FUNCTION_BLOCK TcoQl355P_v_1_x_x EXTENDS TcoCore.TcoComponent
VAR_INPUT
END_VAR
VAR_OUTPUT
END_VAR
VAR
    {attribute addProperty Name "<#Status#>"}
    _status : TcoQlSeriesSupply_Status_v_1_x_x;
    {attribute addProperty Name "<#Config#>"}
    _config : TcoQlSeriesSupply_Config_v_1_x_x;
    _someTaskIsActive : BOOL;
END_VAR
VAR
    {attribute addProperty Name "<#Get Command#>"}
    _getCommandTask : TcoQlGetCommandTask(THIS^);
    {attribute addProperty Name "<#Set Command#>"}
    _setCommandTask : TcoQlSetCommandTask(THIS^);
    {attribute addProperty Name "<#Restore#>"}
    _restoreTask : TcoCore.TcoTask(THIS^);
END_VAR
VAR
    {attribute 'hide'}
    _sb : TcoCore.StringBuilder;
END_VAR

_getCommandTask(inoConfig := _config, inoStatus := _status);
_setCommandTask(inoConfig := _config, inoStatus := _status);
//*************RESTORE********************
_restoreTask.Enabled := TRUE;

IF _restoreTask.Execute() THEN
    Restore();
    _restoreTask.DoneWhen(TRUE);
    _status.ActionDescription := 'Restored';
END_IF
//****************************************

(*~
    <docu>
        <summary>
            Gets the configuration of the IRC 5.
        </summary>
    </docu>
~*)
PROPERTY Config : REFERENCE TO TcoQlSeriesSupply_Config_v_1_x_x
GET
Config REF= _config;
END_GET
END_PROPERTY

METHOD FB_init : BOOL
VAR_INPUT
    bInitRetains : BOOL; // if TRUE, the retain variables are initialized (warm start / cold start)
    bInCopyCode : BOOL; // if TRUE, the instance afterwards gets moved into the copy code (online change)
    ParentObject : ITcoObject;
END_VAR
END_METHOD

METHOD PUBLIC GetCommand : TcoCore.ITcoTaskStatus
VAR_INPUT
    inCommand : TcoQlSeriesSupply_getControl_v_1_x_x;
END_VAR
GetCommand := _getCommandTask.WithParams(inCommand).Invoke();
END_METHOD

PROPERTY GetCommandTask : TcoCore.ITcoTaskStatus
GET
GetCommandTask := _getCommandTask;
END_GET
END_PROPERTY

METHOD PUBLIC GetCurrent : TcoCore.ITcoTaskStatus
VAR_INPUT
    (*~
    <docu>
        <summary>
            The number of the output or status register to which the command relates.
            Note that on single output supplies <N>=1 always.
            Note also that <N>= 3 refers to the AUX output. The AUX output has limited remote control functionality.
            For clarity, the commands where <N>= 3 can be used are explicitly commented; elsewhere only <N>= 1 or <N>= 2 can be used.
        </summary>
    </docu>
    ~*)
    inNValue : USINT;
END_VAR
VAR_OUTPUT
    outCurrent : REAL;
END_VAR
VAR
    command : TcoQlSeriesSupply_GetControl_v_1_x_x;
END_VAR
outCurrent := 0;
command.Command := eTcoQWlSeriesSupplyGetCommands_v_1_x_x.i;
command.NValue := inNValue;
GetCurrent := GetCommand(inCommand := command);

IF GetCurrent.Done THEN
    outCurrent := Status.State.Nr2Value;
END_IF
END_METHOD

METHOD PUBLIC GetOutputIsOff : TcoCore.ITcoTaskStatus
VAR_INPUT
    (*~
    <docu>
        <summary>
            The number of the output or status register to which the command relates.
            Note that on single output supplies <N>=1 always.
            Note also that <N>= 3 refers to the AUX output. The AUX output has limited remote control functionality.
            For clarity, the commands where <N>= 3 can be used are explicitly commented; elsewhere only <N>= 1 or <N>= 2 can be used.
        </summary>
    </docu>
    ~*)
    inNValue : USINT;
END_VAR
VAR_OUTPUT
    outIsOff : BOOL;
END_VAR
VAR
    command : TcoQlSeriesSupply_GetControl_v_1_x_x;
END_VAR
outIsOff := FALSE;
command.Command := eTcoQWlSeriesSupplyGetCommands_v_1_x_x.OP;
command.NValue := inNValue;
GetOutputIsOff := GetCommand(inCommand := command);

IF GetOutputIsOff.Done THEN
    outIsOff := Status.State.Nr2Value = 0;
END_IF
END_METHOD

METHOD PUBLIC GetOutputIsOn : TcoCore.ITcoTaskStatus
VAR_INPUT
    (*~
    <docu>
        <summary>
            The number of the output or status register to which the command relates.
            Note that on single output supplies <N>=1 always.
            Note also that <N>= 3 refers to the AUX output. The AUX output has limited remote control functionality.
            For clarity, the commands where <N>= 3 can be used are explicitly commented; elsewhere only <N>= 1 or <N>= 2 can be used.
        </summary>
    </docu>
    ~*)
    inNValue : USINT;
END_VAR
VAR_OUTPUT
    outIsOn : BOOL;
END_VAR
VAR
    command : TcoQlSeriesSupply_GetControl_v_1_x_x;
END_VAR
outIsOn := FALSE;
command.Command := eTcoQWlSeriesSupplyGetCommands_v_1_x_x.OP;
command.NValue := inNValue;
GetOutputIsOn := GetCommand(inCommand := command);

IF GetOutputIsOn.Done THEN
    outIsOn := Status.State.Nr2Value = 1;
END_IF
END_METHOD

METHOD PUBLIC GetVoltage : TcoCore.ITcoTaskStatus
VAR_INPUT
    (*~
    <docu>
        <summary>
            The number of the output or status register to which the command relates.
            Note that on single output supplies <N>=1 always.
            Note also that <N>= 3 refers to the AUX output. The AUX output has limited remote control functionality.
            For clarity, the commands where <N>= 3 can be used are explicitly commented; elsewhere only <N>= 1 or <N>= 2 can be used.
        </summary>
    </docu>
    ~*)
    inNValue : USINT;
END_VAR
VAR_OUTPUT
    outVoltage : REAL;
END_VAR
VAR
    command : TcoQlSeriesSupply_GetControl_v_1_x_x;
END_VAR
outVoltage := 0;
command.Command := eTcoQWlSeriesSupplyGetCommands_v_1_x_x.V;
command.NValue := inNValue;
GetVoltage := GetCommand(inCommand := command);

IF GetVoltage.Done THEN
    outVoltage := Status.State.Nr2Value;
END_IF
END_METHOD

(*~
    <docu>
        <summary>
            Restores this instance to the Ready state. Can be called explicitly or from within one of the restore mechanisms.
        </summary>
    </docu>
~*)
METHOD Restore : ITcoRestorable
RestoreTasks();
END_METHOD

METHOD INTERNAL RestoreTasks
_getCommandTask.Restore();
_setCommandTask.Restore();
END_METHOD

(*~
    <docu>
        <summary>
            Custom service (manual, maintenance) logic.
            This method must be implemented in derived class.
        </summary>
    </docu>
~*)
METHOD PROTECTED ServiceMode
END_METHOD

METHOD PUBLIC SetCommand : TcoCore.ITcoTaskStatus
VAR_INPUT
    inCommand : TcoQlSeriesSupply_SetControl_v_1_x_x;
END_VAR
SetCommand := _setCommandTask.WithParams(inCommand).Invoke();
END_METHOD

PROPERTY SetCommandTask : TcoCore.ITcoTaskStatus
GET
SetCommandTask := _setCommandTask;
END_GET
END_PROPERTY

METHOD PUBLIC SetCurrent : TcoCore.ITcoTaskStatus
VAR_INPUT
    inCurrent : REAL;
    (*~
    <docu>
        <summary>
            The number of the output or status register to which the command relates.
            Note that on single output supplies <N>=1 always.
            Note also that <N>= 3 refers to the AUX output. The AUX output has limited remote control functionality.
            For clarity, the commands where <N>= 3 can be used are explicitly commented; elsewhere only <N>= 1 or <N>= 2 can be used.
        </summary>
    </docu>
    ~*)
    inNValue : USINT;
END_VAR
VAR
    command : TcoQlSeriesSupply_SetControl_v_1_x_x;
END_VAR
command.Command := eTcoQWlSeriesSupplySetCommands_v_1_x_x.I;
command.NValue := inNValue;
command.NrfValue := inCurrent;
SetCurrent := SetCommand(inCommand := command);
END_METHOD

METHOD PUBLIC SetOutputOff : TcoCore.ITcoTaskStatus
VAR_INPUT
    (*~
    <docu>
        <summary>
            The number of the output or status register to which the command relates.
            Note that on single output supplies <N>=1 always.
            Note also that <N>= 3 refers to the AUX output. The AUX output has limited remote control functionality.
            For clarity, the commands where <N>= 3 can be used are explicitly commented; elsewhere only <N>= 1 or <N>= 2 can be used.
        </summary>
    </docu>
    ~*)
    inNValue : USINT;
END_VAR
VAR
    command : TcoQlSeriesSupply_SetControl_v_1_x_x;
END_VAR
command.Command := eTcoQWlSeriesSupplySetCommands_v_1_x_x.OP;
command.NValue := inNValue;
command.NrfValue := 0;
SetOutputOff := SetCommand(inCommand := command);
END_METHOD

METHOD PUBLIC SetOutputOn : TcoCore.ITcoTaskStatus
VAR_INPUT
    (*~
    <docu>
        <summary>
            The number of the output or status register to which the command relates.
            Note that on single output supplies <N>=1 always.
            Note also that <N>= 3 refers to the AUX output. The AUX output has limited remote control functionality.
            For clarity, the commands where <N>= 3 can be used are explicitly commented; elsewhere only <N>= 1 or <N>= 2 can be used.
        </summary>
    </docu>
    ~*)
    inNValue : USINT;
END_VAR
VAR
    command : TcoQlSeriesSupply_SetControl_v_1_x_x;
END_VAR
command.Command := eTcoQWlSeriesSupplySetCommands_v_1_x_x.OP;
command.NValue := inNValue;
command.NrfValue := 1;
SetOutputOn := SetCommand(inCommand := command);
END_METHOD

METHOD PUBLIC SetVoltage : TcoCore.ITcoTaskStatus
VAR_INPUT
    inVoltage : REAL;
    (*~
    <docu>
        <summary>
            The number of the output or status register to which the command relates.
            Note that on single output supplies <N>=1 always.
            Note also that <N>= 3 refers to the AUX output. The AUX output has limited remote control functionality.
            For clarity, the commands where <N>= 3 can be used are explicitly commented; elsewhere only <N>= 1 or <N>= 2 can be used.
        </summary>
    </docu>
    ~*)
    inNValue : USINT;
END_VAR
VAR
    command : TcoQlSeriesSupply_SetControl_v_1_x_x;
END_VAR
command.Command := eTcoQWlSeriesSupplySetCommands_v_1_x_x.V;
command.NValue := inNValue;
command.NrfValue := inVoltage;
SetVoltage := SetCommand(inCommand := command);
END_METHOD

(*~
    <docu>
        <summary>
            Gets the status of the components.
        </summary>
    </docu>
~*)
PROPERTY Status : REFERENCE TO TcoQlSeriesSupply_Status_v_1_x_x
GET
Status REF= _status;
END_GET
END_PROPERTY

END_FUNCTION_BLOCK

(* stored: Version 1.1.0.1, ProductVersion 3.1.4024.12
   POU TcoQl355P_v_1_x_x: Id {3351a7f4-e4f1-04e8-3ae3-ec074b015e29}, SpecialFunc None
   Folder Operations: Id {e8b663f1-a9d8-0c21-2683-e7c53ff03299}
   Folder Common: Id {c64fa824-d5e6-0c5f-3eca-9b18c97a84ef}
   Folder Generic: Id {0fa8a0b2-76c5-06be-2a99-52e67203b4f2}
   Folder Task: Id {1344c1b8-175a-02e2-1845-1a8160c3a7e2}
   Property Config: Id {0d394bbf-cc1c-00b2-245b-f6a4450329ff}
   Get Get: Id {33cb4413-958b-0fea-2390-664c9ed1d18d}
   Method FB_init: Id {4b8fcfca-d923-0cb6-3a56-bb8a33d6e82e}
   Method GetCommand: Id {35ec3a2d-8699-088d-10ef-6b2159e77b4c}
   Property GetCommandTask: Id {e346ab33-8a9a-0ff9-2fb2-e1ab6d055417}
   Get Get: Id {ceb4c0e1-5052-02c1-1c87-038ae820f955}
   Method GetCurrent: Id {ba6c7d04-667c-0e95-3448-f9bb8eda89bb}
   Method GetOutputIsOff: Id {e968a5b2-fa28-0d5c-3b64-b5eefa949a1a}
   Method GetOutputIsOn: Id {64b4ff7a-12c4-0470-0a9e-d7c6710f1cdf}
   Method GetVoltage: Id {7c7e5362-3d05-026d-0323-0042ae5c5c29}
   Method Restore: Id {1ec27197-5427-0672-1611-f2acf08d391e}
   Method RestoreTasks: Id {c3387e7c-355a-01ce-0d66-89c8a763a695}
   Method ServiceMode: Id {cd2e86cc-91dc-0db1-0291-9006d9ac836e}
   Method SetCommand: Id {e62ff0aa-6a20-0e6f-0576-73a9ca2a0ac5}
   Property SetCommandTask: Id {21ce3437-63d3-0c82-3862-eb42ebd61b67}
   Get Get: Id {858be8ab-d4a7-0feb-24c2-89f2d85cbe57}
   Method SetCurrent: Id {f95506f9-9fc9-0eaf-3be0-a3ceb792c9b3}
   Method SetOutputOff: Id {b26455cd-694a-0b9b-0807-30e3d64e4b48}
   Method SetOutputOn: Id {c3d7ecf8-26aa-0520-3c5f-0ce370da2941}
   Method SetVoltage: Id {74d1228e-8c5e-04da-1b2b-c71026f5b0d6}
   Property Status: Id {a9200237-e208-0004-1b98-3d6bca21b7ff}
   Get Get: Id {62c3e7b1-5416-07c9-1a04-46747a4aecb4} *)
